PROGRAM PRG_LVCP1_Group10
VAR
    // Function Block Instance
    fbContactor: FB_ContactorControl;

    // Contactor 1 IO Structure  
    stContactor_IO: ST_ContactorIO;
    
    // Başlangıç konfigürasyonu için flag
    bContactorInitDone: BOOL := FALSE;
    bCapacitorInitDone: BOOL := FALSE;	
END_VAR



	M_Contactor();
	
	M_Capacitor();

METHOD M_Capacitor : BOOL
VAR
    nGroupIndex : INT;
END_VAR

nGroupIndex := 9;  // Grup 10 için index

IF NOT bCapacitorInitDone THEN
    // Grup 10 değerlerini ata
    GVL_LVCP1.astCompensationGroups[nGroupIndex].rPower := 12.5;
    GVL_LVCP1.astCompensationGroups[nGroupIndex].rVoltage := 450.0;
    GVL_LVCP1.astCompensationGroups[nGroupIndex].nQuantity := 1;
    GVL_LVCP1.astCompensationGroups[nGroupIndex].sTagPrefix := '+EP6-43C1';
    GVL_LVCP1.astCompensationGroups[nGroupIndex].sProductCode := 'ENT.CXD-450-12.5';
    
    bCapacitorInitDone := TRUE;
END_IF

// Grup 10 aktif durumu
GVL_LVCP1.abGroupActive[nGroupIndex] := stContactor_IO.bFeedback;

M_Capacitor := TRUE;
END_METHOD

METHOD M_Contactor : BOOL
VAR_INPUT
END_VAR
IF NOT bContactorInitDone THEN
    // Konfigürasyon parametreleri
    GVL_LVCP1.stGroup10_ContactorHMI.stConfig.sProjectCode := '+EP6-42K1';
    GVL_LVCP1.stGroup10_ContactorHMI.stConfig.sProductCode := 'SCH LC1G115LSEA';
    GVL_LVCP1.stGroup10_ContactorHMI.stConfig.rRatedCurrent := 115.0;
    GVL_LVCP1.stGroup10_ContactorHMI.stConfig.rRatedVoltage := 1000.0;
    GVL_LVCP1.stGroup10_ContactorHMI.stConfig.nPhaseCount := 3;
    GVL_LVCP1.stGroup10_ContactorHMI.stConfig.tFeedbackDelay := T#500MS;
    GVL_LVCP1.stGroup10_ContactorHMI.stConfig.tWeldedDelay := T#2S;
    GVL_LVCP1.stGroup10_ContactorHMI.stConfig.dwOperationLimit := 100000;
    
    // Başlangıç bakım sayacı
    GVL_LVCP1.stGroup10_ContactorHMI.stStatistics.dwRemainingOperations := GVL_LVCP1.stGroup10_ContactorHMI.stConfig.dwOperationLimit;
    
    bContactorInitDone := TRUE;
END_IF

// Function Block Çağrısı
fbContactor(
    // Fiziksel Girişler
    bFeedback := stContactor_IO.bFeedback,
    bPLCControl := stContactor_IO.bPLCControl,
    
    // Güvenlik Girişleri
    bSafetyLoop := GVL_Alarm.bSafetyLoop,
    bInterlock := FALSE,
    
    // Sistem Girişleri
    bMasterReset := GVL_Alarm.bMasterReset,
    
    // HMI Bağlantısı
    stHMI := GVL_LVCP1.stGroup10_ContactorHMI,
    
    // Fiziksel Çıkış
    bOutput => stContactor_IO.bOutput
);

M_Contactor := TRUE;
END_METHOD

END_PROGRAM

(* stored: Version 1.1.0.1, ProductVersion 3.1.4024.15
   POU PRG_LVCP1_Group10: Id {38f25a11-0400-4034-b5c0-0e24df4da03d}, SpecialFunc None
   Method M_Capacitor: Id {4a798277-1514-48cb-927f-3463933bf5c2}
   Method M_Contactor: Id {085c4b52-4ca3-45b4-9e4c-a63e25a20682} *)
